{attribute addProperty BoxType "EL3318-0000-0016"}
{attribute addProperty Id "StatusAT %I*Status_F710A6139311.6251ValueAT %I*INT16217"}
{attribute addProperty CRC "2306082580"}
{attribute addProperty SizeInBites "109"}
{attribute addProperty SizeInBytes "13.625"}
TYPE TC_Channel_89740714 :
STRUCT
	{attribute addProperty Name "Status"}
	Status AT %I* : Status_F710A613;
	{attribute addProperty Name "Value"}
	Value AT %I* : INT;
END_STRUCT
END_TYPE

(* stored: Version 1.2.0.0, ProductVersion 3.1.4024.9
   DUT TC_Channel_89740714: Id {be8a44d6-b826-4ca8-b7b7-ca623d7e92cc} *)
